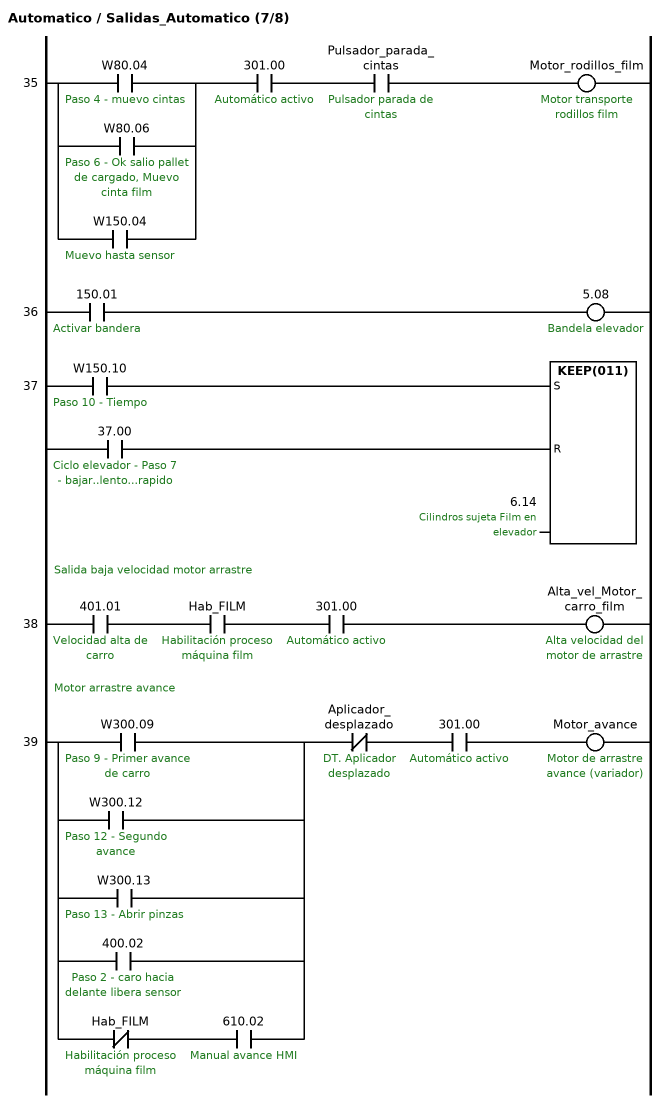
; [picture p72: Automatico / Salidas_Automatico, rungs 35-39]
; rung 35
LD W80.04  ; Paso 4 - muevo cintas
OR W80.06  ; Paso 6 - Ok salio pallet de cargado, Muevo cinta film
OR W150.04  ; Muevo hasta sensor
AND 301.00  ; Automático activo
AND Pulsador_parada_cintas  ; Pulsador parada de cintas
OUT Motor_rodillos_film  ; Motor transporte rodillos film
; rung 36
LD 150.01  ; Activar bandera
OUT 5.08  ; Bandela elevador
; rung 37
LD W150.10  ; Paso 10 - Tiempo
LD 37.00  ; Ciclo elevador - Paso 7 - bajar..lento...rapido
KEEP(011) 6.14  ; Cilindros sujeta Film en elevador
; rung 38: Salida baja velocidad motor arrastre
LD 401.01  ; Velocidad alta de carro
AND Hab_FILM  ; Habilitación proceso máquina film
AND 301.00  ; Automático activo
OUT Alta_vel_Motor_carro_film  ; Alta velocidad del motor de arrastre
; rung 39: Motor arrastre avance
LD W300.09  ; Paso 9 - Primer avance de carro
OR W300.12  ; Paso 12 - Segundo avance
OR W300.13  ; Paso 13 - Abrir pinzas
OR 400.02  ; Paso 2 - caro hacia delante libera sensor
LDNOT Hab_FILM  ; Habilitación proceso máquina film
AND 610.02  ; Manual avance HMI
ORLD
ANDNOT Aplicador_desplazado  ; DT. Aplicador desplazado
AND 301.00  ; Automático activo
OUT Motor_avance  ; Motor de arrastre avance (variador)

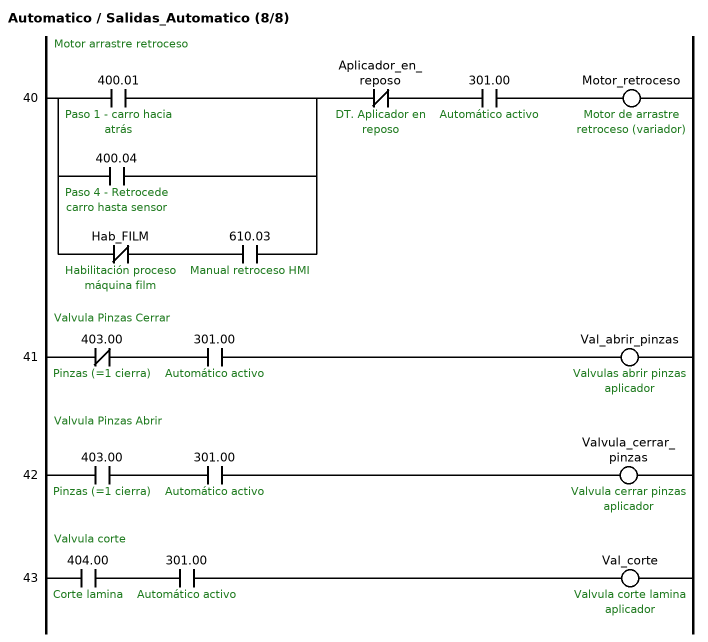
; rung 40: Motor arrastre retroceso
LD 400.01  ; Paso 1 - carro hacia atrás
OR 400.04  ; Paso 4 - Retrocede carro hasta sensor
LDNOT Hab_FILM  ; Habilitación proceso máquina film
AND 610.03  ; Manual retroceso HMI
ORLD
ANDNOT Aplicador_en_reposo  ; DT. Aplicador en reposo
AND 301.00  ; Automático activo
OUT Motor_retroceso  ; Motor de arrastre retroceso (variador)
; rung 41: Valvula Pinzas Cerrar
LDNOT 403.00  ; Pinzas (=1 cierra)
AND 301.00  ; Automático activo
OUT Val_abrir_pinzas  ; Valvulas abrir pinzas aplicador
; rung 42: Valvula Pinzas Abrir
LD 403.00  ; Pinzas (=1 cierra)
AND 301.00  ; Automático activo
OUT Valvula_cerrar_pinzas  ; Valvula cerrar pinzas aplicador
; rung 43: Valvula corte
LD 404.00  ; Corte lamina
AND 301.00  ; Automático activo
OUT Val_corte  ; Valvula corte lamina aplicador

### Section END
; rung 0
END(001)

## Program Manuales (cyclic task 2)
Local symbols
OLD_M976 BOOL
r REAL

### Section Manuales

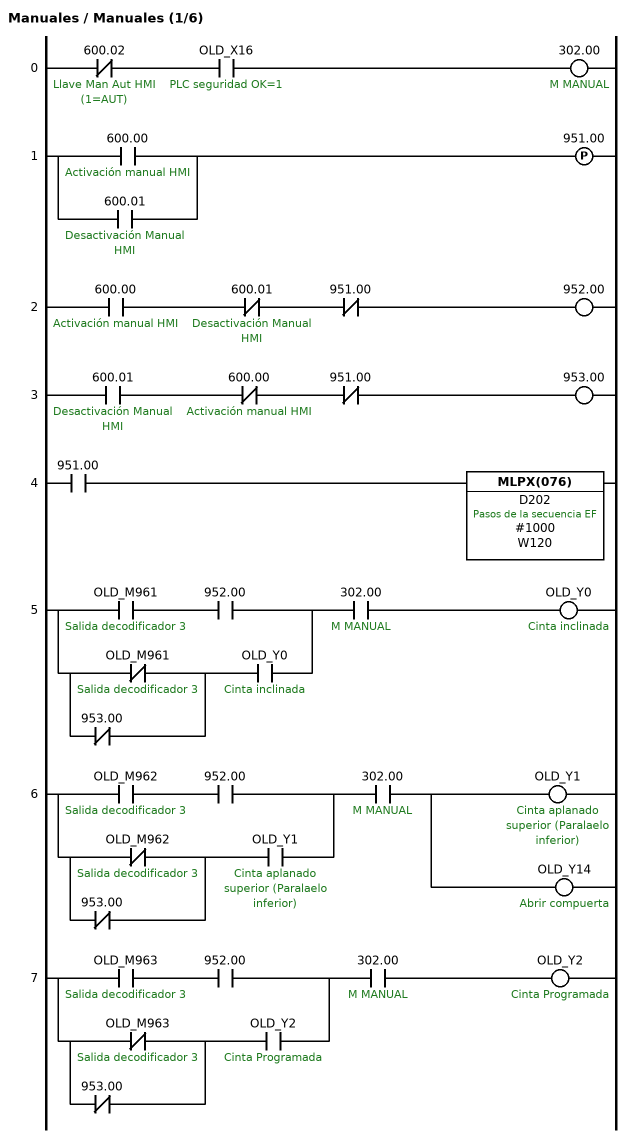
; rung 0
LDNOT 600.02  ; Llave Man Aut HMI (1=AUT)
AND OLD_X16  ; PLC seguridad OK=1
OUT 302.00  ; M MANUAL
; rung 1
LD 600.00  ; Activación manual HMI
OR 600.01  ; Desactivación Manual HMI
DIFU(013) 951.00
; rung 2
LD 600.00  ; Activación manual HMI
ANDNOT 600.01  ; Desactivación Manual HMI
ANDNOT 951.00
OUT 952.00
; rung 3
LD 600.01  ; Desactivación Manual HMI
ANDNOT 600.00  ; Activación manual HMI
ANDNOT 951.00
OUT 953.00
; rung 4
LD 951.00
MLPX(076) D202 #1000 W120  ; Pasos de la secuencia EF
; rung 5
LD OLD_M961  ; Salida decodificador 3
AND 952.00
LDNOT OLD_M961  ; Salida decodificador 3
ORNOT 953.00
AND OLD_Y0  ; Cinta inclinada
ORLD
AND 302.00  ; M MANUAL
OUT OLD_Y0  ; Cinta inclinada
; rung 6
LD OLD_M962  ; Salida decodificador 3
AND 952.00
LDNOT OLD_M962  ; Salida decodificador 3
ORNOT 953.00
AND OLD_Y1  ; Cinta aplanado superior (Paralaelo inferior)
ORLD
AND 302.00  ; M MANUAL
OUT OLD_Y1  ; Cinta aplanado superior (Paralaelo inferior)
OUT OLD_Y14  ; Abrir compuerta
; rung 7
LD OLD_M963  ; Salida decodificador 3
AND 952.00
LDNOT OLD_M963  ; Salida decodificador 3
ORNOT 953.00
AND OLD_Y2  ; Cinta Programada
ORLD
AND 302.00  ; M MANUAL
OUT OLD_Y2  ; Cinta Programada

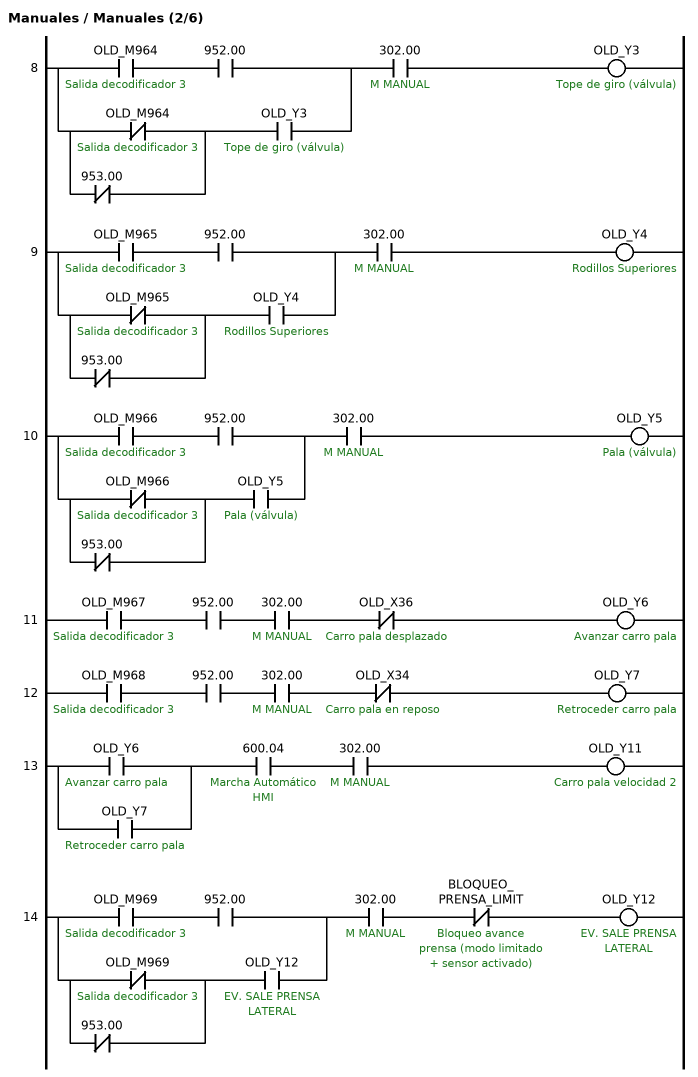
; rung 8
LD OLD_M964  ; Salida decodificador 3
AND 952.00
LDNOT OLD_M964  ; Salida decodificador 3
ORNOT 953.00
AND OLD_Y3  ; Tope de giro (válvula)
ORLD
AND 302.00  ; M MANUAL
OUT OLD_Y3  ; Tope de giro (válvula)
; rung 9
LD OLD_M965  ; Salida decodificador 3
AND 952.00
LDNOT OLD_M965  ; Salida decodificador 3
ORNOT 953.00
AND OLD_Y4  ; Rodillos Superiores
ORLD
AND 302.00  ; M MANUAL
OUT OLD_Y4  ; Rodillos Superiores
; rung 10
LD OLD_M966  ; Salida decodificador 3
AND 952.00
LDNOT OLD_M966  ; Salida decodificador 3
ORNOT 953.00
AND OLD_Y5  ; Pala (válvula)
ORLD
AND 302.00  ; M MANUAL
OUT OLD_Y5  ; Pala (válvula)
; rung 11
LD OLD_M967  ; Salida decodificador 3
AND 952.00
AND 302.00  ; M MANUAL
ANDNOT OLD_X36  ; Carro pala desplazado
OUT OLD_Y6  ; Avanzar carro pala
; rung 12
LD OLD_M968  ; Salida decodificador 3
AND 952.00
AND 302.00  ; M MANUAL
ANDNOT OLD_X34  ; Carro pala en reposo
OUT OLD_Y7  ; Retroceder carro pala
; rung 13
LD OLD_Y6  ; Avanzar carro pala
OR OLD_Y7  ; Retroceder carro pala
AND 600.04  ; Marcha Automático HMI
AND 302.00  ; M MANUAL
OUT OLD_Y11  ; Carro pala velocidad 2
; rung 14
LD OLD_M969  ; Salida decodificador 3
AND 952.00
LDNOT OLD_M969  ; Salida decodificador 3
ORNOT 953.00
AND OLD_Y12  ; EV. SALE PRENSA LATERAL
ORLD
AND 302.00  ; M MANUAL
ANDNOT BLOQUEO_PRENSA_LIMIT  ; Bloqueo avance prensa (modo limitado + sensor activado)
OUT OLD_Y12  ; EV. SALE PRENSA LATERAL

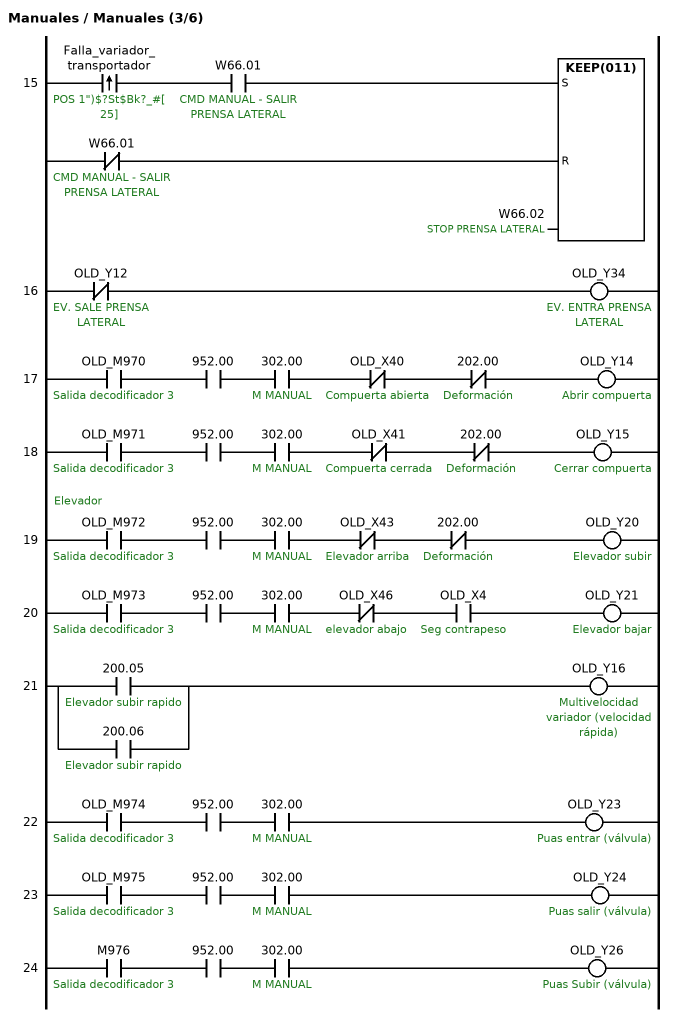
; rung 15
@LD Falla_variador_transportador  ; POS 1")$?St$Bk?_#[25]
AND W66.01  ; CMD MANUAL - SALIR PRENSA LATERAL
LDNOT W66.01  ; CMD MANUAL - SALIR PRENSA LATERAL
KEEP(011) W66.02  ; STOP PRENSA LATERAL
; rung 16
LDNOT OLD_Y12  ; EV. SALE PRENSA LATERAL
OUT OLD_Y34  ; EV. ENTRA PRENSA LATERAL
; rung 17
LD OLD_M970  ; Salida decodificador 3
AND 952.00
AND 302.00  ; M MANUAL
ANDNOT OLD_X40  ; Compuerta abierta
ANDNOT 202.00  ; Deformación
OUT OLD_Y14  ; Abrir compuerta
; rung 18
LD OLD_M971  ; Salida decodificador 3
AND 952.00
AND 302.00  ; M MANUAL
ANDNOT OLD_X41  ; Compuerta cerrada
ANDNOT 202.00  ; Deformación
OUT OLD_Y15  ; Cerrar compuerta
; rung 19: Elevador
LD OLD_M972  ; Salida decodificador 3
AND 952.00
AND 302.00  ; M MANUAL
ANDNOT OLD_X43  ; Elevador arriba
ANDNOT 202.00  ; Deformación
OUT OLD_Y20  ; Elevador subir
; rung 20
LD OLD_M973  ; Salida decodificador 3
AND 952.00
AND 302.00  ; M MANUAL
ANDNOT OLD_X46  ; elevador abajo
AND OLD_X4  ; Seg contrapeso
OUT OLD_Y21  ; Elevador bajar
; rung 21
LD 200.05  ; Elevador subir rapido
OR 200.06  ; Elevador subir rapido
OUT OLD_Y16  ; Multivelocidad variador (velocidad rápida)
; rung 22
LD OLD_M974  ; Salida decodificador 3
AND 952.00
AND 302.00  ; M MANUAL
OUT OLD_Y23  ; Puas entrar (válvula)
; rung 23
LD OLD_M975  ; Salida decodificador 3
AND 952.00
AND 302.00  ; M MANUAL
OUT OLD_Y24  ; Puas salir (válvula)
; rung 24
LD M976  ; Salida decodificador 3
AND 952.00
AND 302.00  ; M MANUAL
OUT OLD_Y26  ; Puas Subir (válvula)

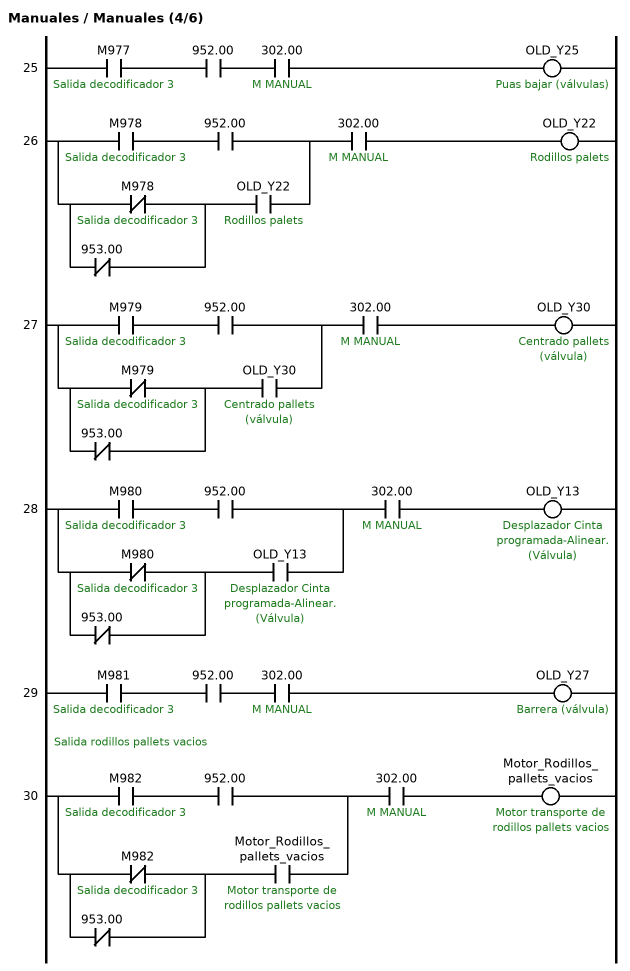
; rung 25
LD M977  ; Salida decodificador 3
AND 952.00
AND 302.00  ; M MANUAL
OUT OLD_Y25  ; Puas bajar (válvulas)
; rung 26
LD M978  ; Salida decodificador 3
AND 952.00
LDNOT M978  ; Salida decodificador 3
ORNOT 953.00
AND OLD_Y22  ; Rodillos palets
ORLD
AND 302.00  ; M MANUAL
OUT OLD_Y22  ; Rodillos palets
; rung 27
LD M979  ; Salida decodificador 3
AND 952.00
LDNOT M979  ; Salida decodificador 3
ORNOT 953.00
AND OLD_Y30  ; Centrado pallets (válvula)
ORLD
AND 302.00  ; M MANUAL
OUT OLD_Y30  ; Centrado pallets (válvula)
; rung 28
LD M980  ; Salida decodificador 3
AND 952.00
LDNOT M980  ; Salida decodificador 3
ORNOT 953.00
AND OLD_Y13  ; Desplazador Cinta programada-Alinear. (Válvula)
ORLD
AND 302.00  ; M MANUAL
OUT OLD_Y13  ; Desplazador Cinta programada-Alinear. (Válvula)
; rung 29
LD M981  ; Salida decodificador 3
AND 952.00
AND 302.00  ; M MANUAL
OUT OLD_Y27  ; Barrera (válvula)
; rung 30: Salida rodillos pallets vacios
LD M982  ; Salida decodificador 3
AND 952.00
LDNOT M982  ; Salida decodificador 3
ORNOT 953.00
AND Motor_Rodillos_pallets_vacios  ; Motor transporte de rodillos pallets vacios
ORLD
AND 302.00  ; M MANUAL
OUT Motor_Rodillos_pallets_vacios  ; Motor transporte de rodillos pallets vacios

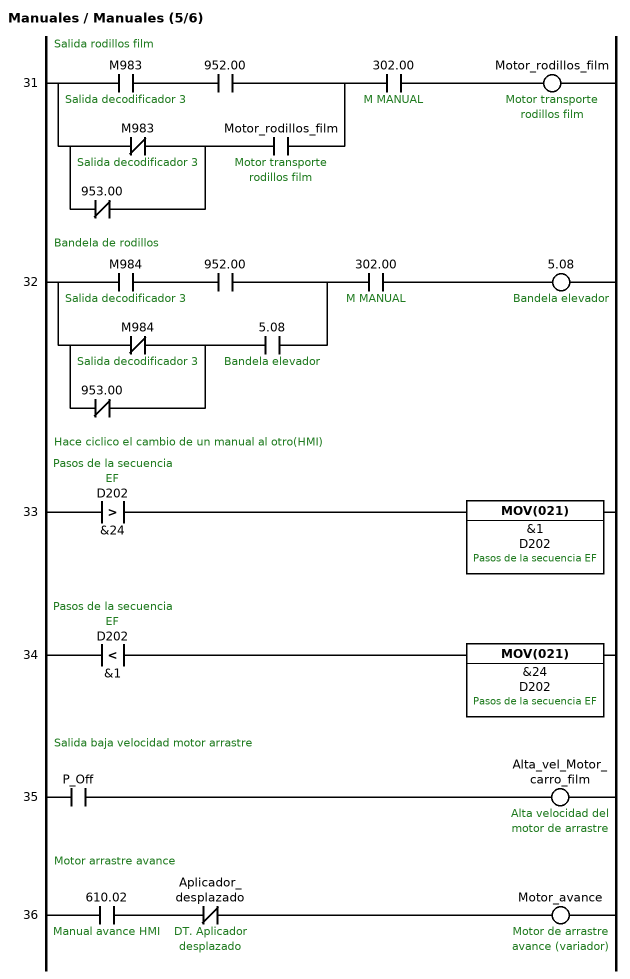
; rung 31: Salida rodillos film
LD M983  ; Salida decodificador 3
AND 952.00
LDNOT M983  ; Salida decodificador 3
ORNOT 953.00
AND Motor_rodillos_film  ; Motor transporte rodillos film
ORLD
AND 302.00  ; M MANUAL
OUT Motor_rodillos_film  ; Motor transporte rodillos film
; rung 32: Bandela de rodillos
LD M984  ; Salida decodificador 3
AND 952.00
LDNOT M984  ; Salida decodificador 3
ORNOT 953.00
AND 5.08  ; Bandela elevador
ORLD
AND 302.00  ; M MANUAL
OUT 5.08  ; Bandela elevador
; rung 33: Hace ciclico el cambio de un manual al otro(HMI)
LD>(320) D202 &24  ; Pasos de la secuencia EF
MOV(021) &1 D202  ; Pasos de la secuencia EF
; rung 34
LD<(310) D202 &1  ; Pasos de la secuencia EF
MOV(021) &24 D202  ; Pasos de la secuencia EF
; rung 35: Salida baja velocidad motor arrastre
LD P_Off
OUT Alta_vel_Motor_carro_film  ; Alta velocidad del motor de arrastre
; rung 36: Motor arrastre avance
LD 610.02  ; Manual avance HMI
ANDNOT Aplicador_desplazado  ; DT. Aplicador desplazado
OUT Motor_avance  ; Motor de arrastre avance (variador)

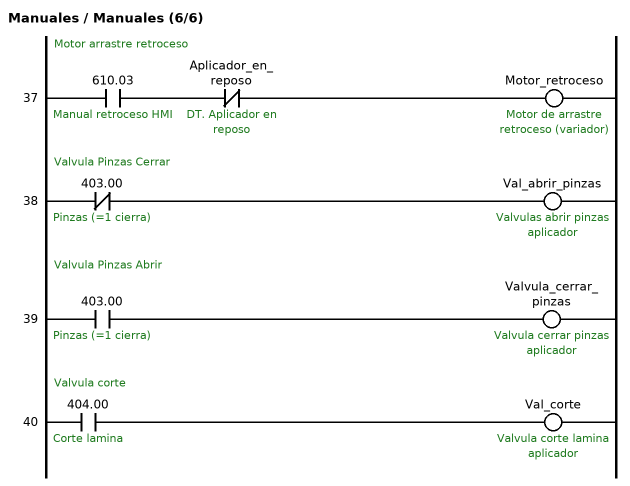
; rung 37: Motor arrastre retroceso
LD 610.03  ; Manual retroceso HMI
ANDNOT Aplicador_en_reposo  ; DT. Aplicador en reposo
OUT Motor_retroceso  ; Motor de arrastre retroceso (variador)
; rung 38: Valvula Pinzas Cerrar
LDNOT 403.00  ; Pinzas (=1 cierra)
OUT Val_abrir_pinzas  ; Valvulas abrir pinzas aplicador
; rung 39: Valvula Pinzas Abrir
LD 403.00  ; Pinzas (=1 cierra)
OUT Valvula_cerrar_pinzas  ; Valvula cerrar pinzas aplicador
; rung 40: Valvula corte
LD 404.00  ; Corte lamina
OUT Val_corte  ; Valvula corte lamina aplicador

### Section END
; rung 0
END(001)

## Function block Conversion_Encoder
VAR_INPUT
  Encoder : DINT;  (* Se coloca el registro de encoder que proviene de un modulo por ejemplo *)
  Constante_conversion : REAL;  (* Constante para conversion en milimetros *)
END_VAR
VAR_OUTPUT
  Encoder_en_mm : DINT;
END_VAR
VAR
  Encoder_real : REAL;
END_VAR
Encoder_real:= DINT_TO_REAL(Encoder);

Encoder_en_mm:=  REAL_TO_DINT(encoder_real*Constante_conversion);

## Function block Funcion_baja_velocidad
VAR_INPUT
  Encoder_mm : UDINT;
  Destino_mm : UDINT;
  Distancia_aproximacion : DINT;
END_VAR
VAR_OUTPUT
  Activa_baja_velocidad : BOOL;
  Activa_alta_velocidad : BOOL;
END_VAR
VAR
  Auxiliar : DINT;
END_VAR
Auxiliar:= UDINT_TO_DINT(Encoder_mm-Destino_mm);

IF Auxiliar < 0 THEN
		Auxiliar:=  Auxiliar*-1;
	END_IF;

IF Auxiliar <= Distancia_aproximacion THEN
		Activa_baja_velocidad:= TRUE;
		Activa_alta_velocidad:= FALSE;
ELSE
       Activa_baja_velocidad:= FALSE;
	   Activa_alta_velocidad:= TRUE;
END_IF;